FUNCTION_BLOCK FB_FIS_MAMDANI
VAR_IN_OUT
	FIS:MAMFIS;
END_VAR
VAR
	i,j: DINT;	
	fbAggregation:FB_AGGREGATION;
END_VAR

//Fuzzufication inteface				
	//Membership degrees calculation 
	FOR i:=1 TO NumOfFISInputs DO
		FOR j:=1 TO FIS.inputs[i].NumberOfMF DO
			FIS.MD[i,j]:= 
				fMembershipDegree(
					CrispInput := FIS.Inputs[i].CrispValue,
					MF:= FIS.Inputs[i].MF[j]);
		END_FOR	 
	END_FOR
//Implication: ImplicationFB is called By FBAggregation

//Aggregation FBis called by Deffuzification function
	fbAggregation.Myrules:=FIS.Rules;
	fbAggregation.MyFISoutputs:=FIS.Outputs;
//Deffuzification
	FIS.Outputs[1].CrispValue:=fCentroid(100,FIS.Outputs[1].Range,fbAggregation);

END_FUNCTION_BLOCK

(* stored: Version 1.1.0.1, ProductVersion 3.1.4024.6
   POU FB_FIS_MAMDANI: Id {5051e573-b6fd-4153-ab29-e97bf2515070}, SpecialFunc None *)
